Omron CX-Programmer project NewProject (CX-Programmer 9.73)

# PLC NewPLC1: CP1E N60

## Global symbols (name address type ; comment)
0 CHANNEL  ; Timer_2
0.00 BOOL  ; Gripper 1 Unclamp
0.01 BOOL  ; Gripper 1 Clamp
0.02 BOOL  ; Gripper 2 Unclamp
0.03 BOOL  ; Gripper 2 Clamp
0.04 BOOL  ; Rotate CCW
0.05 BOOL  ; Rotate CW
0.06 BOOL  ; Cutting  BWD
0.07 BOOL  ; Cutting FWD
0.08 BOOL  ; Detect component
0.09 BOOL  ; Emergency button
0.10 BOOL  ; Reset button
0.11 BOOL  ; Start Button
100.00 BOOL  ; Grip 1 Clamp/Unclamp
100.01 BOOL  ; Grip 2 Clamp/Unclamp
100.02 BOOL  ; Rotate CW/CCW
100.04 BOOL  ; Blow ON
100.05 BOOL  ; Cutting FWD/BWD
101.00 BOOL  ; Relay Wave Bowl
101.01 BOOL  ; TL GREEN
101.02 BOOL  ; TL RED
101.03 BOOL  ; TL YELLOW
1.00 BOOL  ; Pick Finish
1.01 BOOL  ; rotate finish
1.02 BOOL  ; cut finish
1.11 BOOL  ; Auto mode
20 CHANNEL  ; TIMER_02
200.00 BOOL  ; Gripper 1 Unclamp
200.01 BOOL  ; Gripper 1 Clamp
200.02 BOOL  ; Gripper 2 Unclamp
200.03 BOOL  ; Gripper 2 Clamp
200.04 BOOL  ; Rotate CCW
200.05 BOOL  ; Rotate CW
200.06 BOOL  ; Cutting BWD
200.07 BOOL  ; Cutting FWD
200.08 BOOL  ; Detect Comp
201.00 BOOL  ; Gripper 1
201.01 BOOL  ; Gripper 2
201.02 BOOL  ; Rotate
201.03 BOOL  ; Cutting
201.04 BOOL  ; Manual
201.05 BOOL  ; Auto
201.06 BOOL  ; Emg
201.07 BOOL  ; Start Button
201.08 BOOL  ; Reset Button
201.09 BOOL  ; camera capture
202.00 BOOL  ; Cyl Gripper 1 Clamp/Unclamp
202.01 BOOL  ; Cyl Gripper 2 Clamp/Unclamp
202.02 BOOL  ; Cyl Rotate CW/CCW
202.03 BOOL  ; Blow Bowl ON
202.04 BOOL  ; Cyl Cutting FWD/BWD
202.05 BOOL  ; Process ON
202.06 BOOL  ; Relay Wave ON
203.01 BOOL  ; Camera Capture
203.02 BOOL  ; Move Pick
203.03 BOOL  ; Move Pick Finish
203.04 BOOL  ; move pick finish AR
203.05 BOOL  ; Polarity Result
203.06 BOOL  ; Polarity OK
203.07 BOOL  ; Polarity NG
203.08 BOOL  ; Move to cut
203.09 BOOL  ; Move Cut Finish
203.10 BOOL  ; Move to Pick Finish
203.11 BOOL  ; release cutter
203.12 BOOL  ; capture result
203.13 BOOL  ; Move to Rotate
203.14 BOOL  ; Move to rotate finish
203.15 BOOL  ; Move to Cut after rotate
204.00 BOOL  ; Move to cut after rotate finish
204.01 BOOL  ; Rotate release
205.00 BOOL  ; test
206.00 BOOL  ; Gripper 1 Unclamp
206.01 BOOL  ; Gripper 1 Clamp
206.02 BOOL  ; Gripper 2 Unclamp
206.03 BOOL  ; Gripper 2 Clamp
206.04 BOOL  ; Rotate CCW
206.05 BOOL  ; Rotate CW
206.06 BOOL  ; Cutting BWD
206.07 BOOL  ; Cutting FWD
206.08 BOOL  ; M_Out_Blow
206.09 BOOL  ; m_Detect Comp
206.10 BOOL  ; Bowl Feeder
206.11 BOOL  ; EMG
206.12 BOOL  ; RST
207.00 BOOL  ; Grip 1 Clamp
207.01 BOOL  ; Grip 2 clamp
207.02 BOOL  ; Rotate CW CCW
207.03 BOOL  ; Cutting On
207.04 BOOL  ; Blow On
207.05 BOOL  ; Bowl Feeder
209.01 BOOL  ; TRY LAH
210.00 BOOL  ; pick finish
210.01 BOOL  ; rotate finish
210.02 BOOL  ; cut finish
210.03 BOOL  ; pick move
210.04 BOOL  ; stts pick
210.05 BOOL  ; apalah
210.06 BOOL  ; 1
210.07 BOOL  ; 2
210.08 BOOL  ; stts
210.09 BOOL  ; ok
2.00 BOOL  ; Manual mode
4.00 BOOL  ; Gripper 1 Unclamp
T000 BOOL  ; TIMER_01
T002 BOOL  ; TIMER_02
T003 BOOL  ; Release timer

## Program Auto (cyclic task 0)

### Section PC_INTERFACE

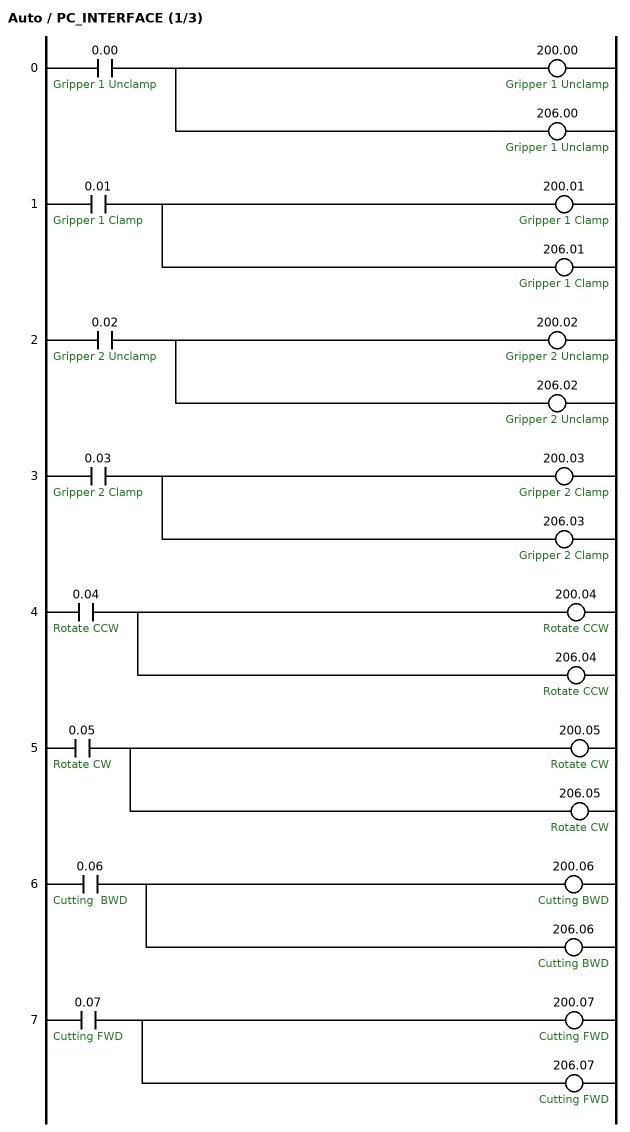
; rung 0
LD 0.00  ; Gripper 1 Unclamp
OUT 200.00  ; Gripper 1 Unclamp
OUT 206.00  ; Gripper 1 Unclamp
; rung 1
LD 0.01  ; Gripper 1 Clamp
OUT 200.01  ; Gripper 1 Clamp
OUT 206.01  ; Gripper 1 Clamp
; rung 2
LD 0.02  ; Gripper 2 Unclamp
OUT 200.02  ; Gripper 2 Unclamp
OUT 206.02  ; Gripper 2 Unclamp
; rung 3
LD 0.03  ; Gripper 2 Clamp
OUT 200.03  ; Gripper 2 Clamp
OUT 206.03  ; Gripper 2 Clamp
; rung 4
LD 0.04  ; Rotate CCW
OUT 200.04  ; Rotate CCW
OUT 206.04  ; Rotate CCW
; rung 5
LD 0.05  ; Rotate CW
OUT 200.05  ; Rotate CW
OUT 206.05  ; Rotate CW
; rung 6
LD 0.06  ; Cutting  BWD
OUT 200.06  ; Cutting BWD
OUT 206.06  ; Cutting BWD
; rung 7
LD 0.07  ; Cutting FWD
OUT 200.07  ; Cutting FWD
OUT 206.07  ; Cutting FWD

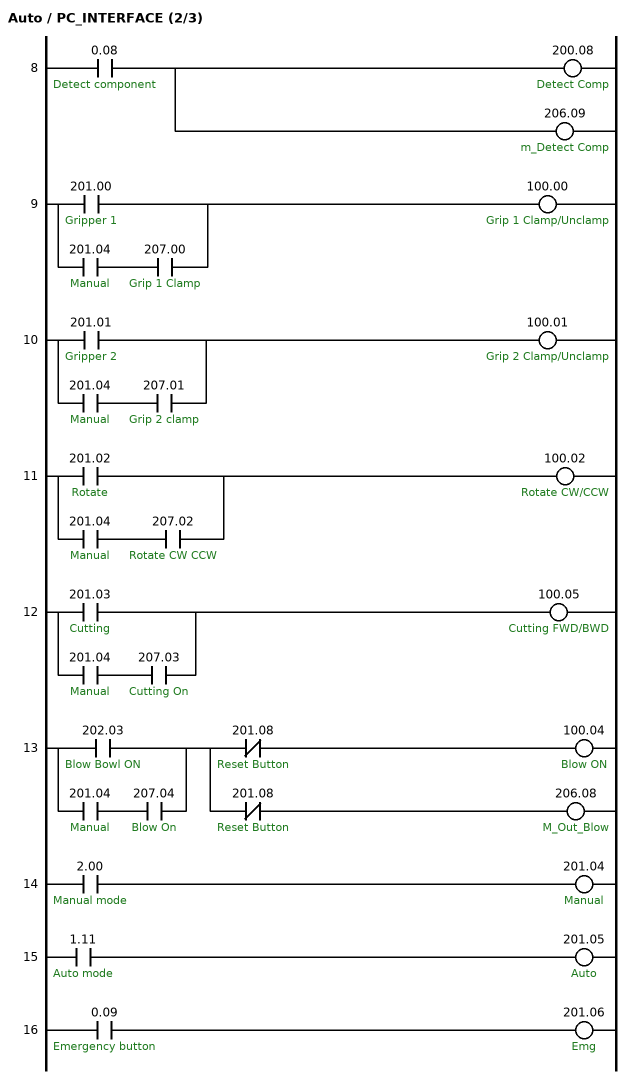
; rung 8
LD 0.08  ; Detect component
OUT 200.08  ; Detect Comp
OUT 206.09  ; m_Detect Comp
; rung 9
LD 201.00  ; Gripper 1
LD 201.04  ; Manual
AND 207.00  ; Grip 1 Clamp
ORLD
OUT 100.00  ; Grip 1 Clamp/Unclamp
; rung 10
LD 201.01  ; Gripper 2
LD 201.04  ; Manual
AND 207.01  ; Grip 2 clamp
ORLD
OUT 100.01  ; Grip 2 Clamp/Unclamp
; rung 11
LD 201.02  ; Rotate
LD 201.04  ; Manual
AND 207.02  ; Rotate CW CCW
ORLD
OUT 100.02  ; Rotate CW/CCW
; rung 12
LD 201.03  ; Cutting
LD 201.04  ; Manual
AND 207.03  ; Cutting On
ORLD
OUT 100.05  ; Cutting FWD/BWD
; rung 13
LD 202.03  ; Blow Bowl ON
LD 201.04  ; Manual
AND 207.04  ; Blow On
ORLD
OUT TR0
ANDNOT 201.08  ; Reset Button
OUT 100.04  ; Blow ON
LD TR0
ANDNOT 201.08  ; Reset Button
OUT 206.08  ; M_Out_Blow
; rung 14
LD 2.00  ; Manual mode
OUT 201.04  ; Manual
; rung 15
LD 1.11  ; Auto mode
OUT 201.05  ; Auto
; rung 16
LD 0.09  ; Emergency button
OUT 201.06  ; Emg

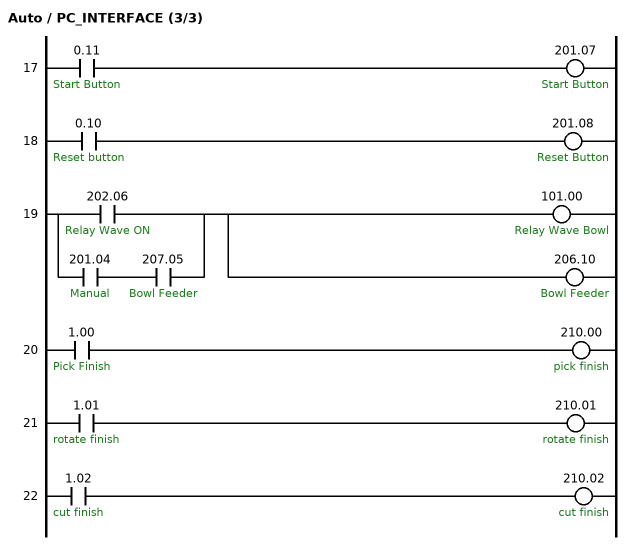
; rung 17
LD 0.11  ; Start Button
OUT 201.07  ; Start Button
; rung 18
LD 0.10  ; Reset button
OUT 201.08  ; Reset Button
; rung 19
LD 202.06  ; Relay Wave ON
LD 201.04  ; Manual
AND 207.05  ; Bowl Feeder
ORLD
OUT 101.00  ; Relay Wave Bowl
OUT 206.10  ; Bowl Feeder
; rung 20
LD 1.00  ; Pick Finish
OUT 210.00  ; pick finish
; rung 21
LD 1.01  ; rotate finish
OUT 210.01  ; rotate finish
; rung 22
LD 1.02  ; cut finish
OUT 210.02  ; cut finish

### Section PROGRAM

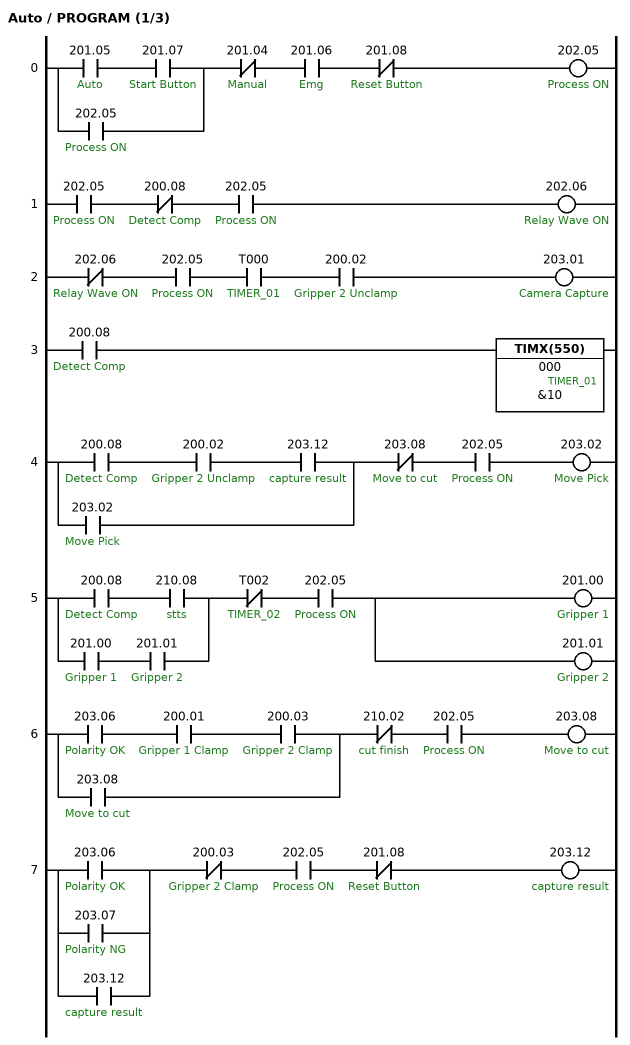
; rung 0
LD 201.05  ; Auto
AND 201.07  ; Start Button
OR 202.05  ; Process ON
ANDNOT 201.04  ; Manual
AND 201.06  ; Emg
ANDNOT 201.08  ; Reset Button
OUT 202.05  ; Process ON
; rung 1
LD 202.05  ; Process ON
ANDNOT 200.08  ; Detect Comp
AND 202.05  ; Process ON
OUT 202.06  ; Relay Wave ON
; rung 2
LDNOT 202.06  ; Relay Wave ON
AND 202.05  ; Process ON
AND T000  ; TIMER_01
AND 200.02  ; Gripper 2 Unclamp
OUT 203.01  ; Camera Capture
; rung 3
LD 200.08  ; Detect Comp
TIMX(550) 000 &10  ; TIMER_01
; rung 4
LD 200.08  ; Detect Comp
AND 200.02  ; Gripper 2 Unclamp
AND 203.12  ; capture result
OR 203.02  ; Move Pick
ANDNOT 203.08  ; Move to cut
AND 202.05  ; Process ON
OUT 203.02  ; Move Pick
; rung 5
LD 200.08  ; Detect Comp
AND 210.08  ; stts
LD 201.00  ; Gripper 1
AND 201.01  ; Gripper 2
ORLD
ANDNOT T002  ; TIMER_02
AND 202.05  ; Process ON
OUT 201.00  ; Gripper 1
OUT 201.01  ; Gripper 2
; rung 6
LD 203.06  ; Polarity OK
AND 200.01  ; Gripper 1 Clamp
AND 200.03  ; Gripper 2 Clamp
OR 203.08  ; Move to cut
ANDNOT 210.02  ; cut finish
AND 202.05  ; Process ON
OUT 203.08  ; Move to cut
; rung 7
LD 203.06  ; Polarity OK
OR 203.07  ; Polarity NG
OR 203.12  ; capture result
ANDNOT 200.03  ; Gripper 2 Clamp
AND 202.05  ; Process ON
ANDNOT 201.08  ; Reset Button
OUT 203.12  ; capture result

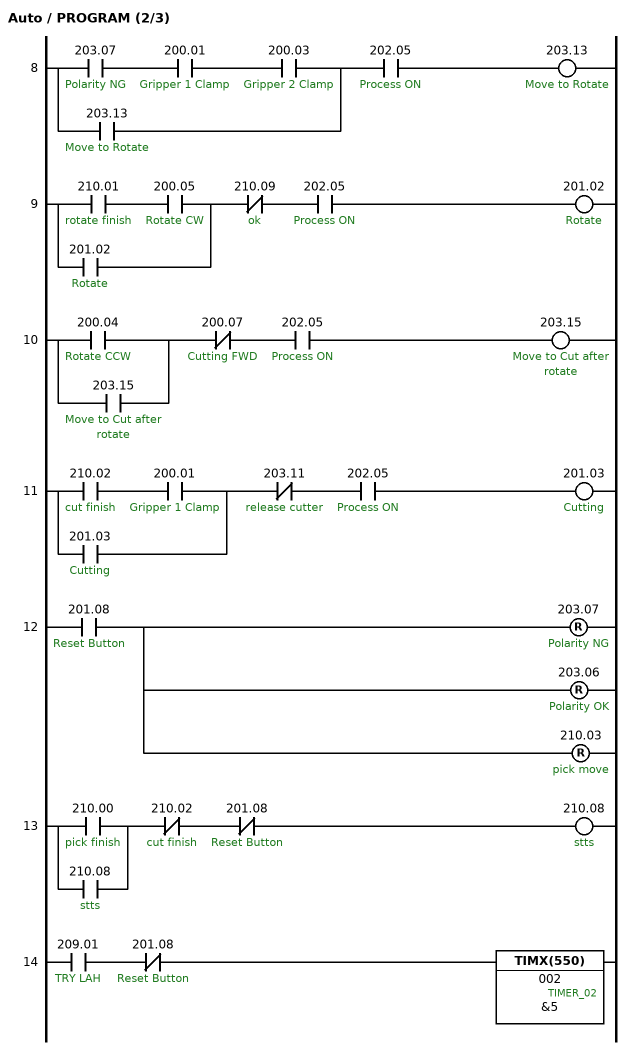
; rung 8
LD 203.07  ; Polarity NG
AND 200.01  ; Gripper 1 Clamp
AND 200.03  ; Gripper 2 Clamp
OR 203.13  ; Move to Rotate
AND 202.05  ; Process ON
OUT 203.13  ; Move to Rotate
; rung 9
LD 210.01  ; rotate finish
AND 200.05  ; Rotate CW
OR 201.02  ; Rotate
ANDNOT 210.09  ; ok
AND 202.05  ; Process ON
OUT 201.02  ; Rotate
; rung 10
LD 200.04  ; Rotate CCW
OR 203.15  ; Move to Cut after rotate
ANDNOT 200.07  ; Cutting FWD
AND 202.05  ; Process ON
OUT 203.15  ; Move to Cut after rotate
; rung 11
LD 210.02  ; cut finish
AND 200.01  ; Gripper 1 Clamp
OR 201.03  ; Cutting
ANDNOT 203.11  ; release cutter
AND 202.05  ; Process ON
OUT 201.03  ; Cutting
; rung 12
LD 201.08  ; Reset Button
RSET 203.07  ; Polarity NG
RSET 203.06  ; Polarity OK
RSET 210.03  ; pick move
; rung 13
LD 210.00  ; pick finish
OR 210.08  ; stts
ANDNOT 210.02  ; cut finish
ANDNOT 201.08  ; Reset Button
OUT 210.08  ; stts
; rung 14
LD 209.01  ; TRY LAH
ANDNOT 201.08  ; Reset Button
TIMX(550) 002 &5  ; TIMER_02

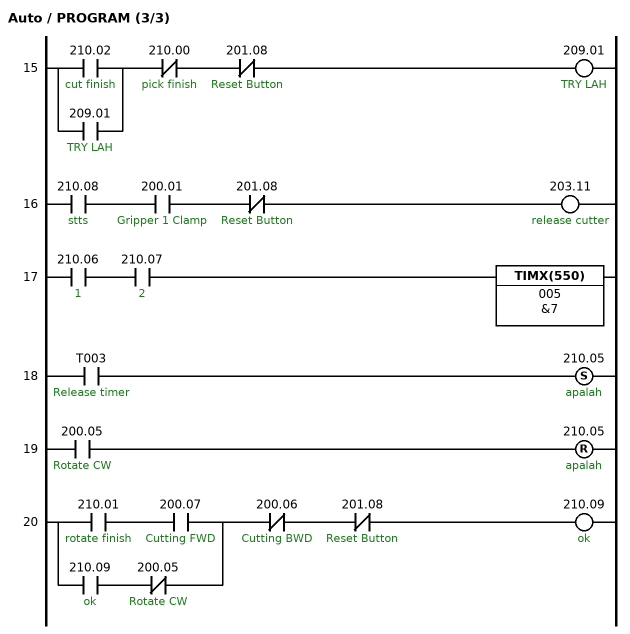
; rung 15
LD 210.02  ; cut finish
OR 209.01  ; TRY LAH
ANDNOT 210.00  ; pick finish
ANDNOT 201.08  ; Reset Button
OUT 209.01  ; TRY LAH
; rung 16
LD 210.08  ; stts
AND 200.01  ; Gripper 1 Clamp
ANDNOT 201.08  ; Reset Button
OUT 203.11  ; release cutter
; rung 17
LD 210.06  ; 1
AND 210.07  ; 2
TIMX(550) 005 &7
; rung 18
LD T003  ; Release timer
SET 210.05  ; apalah
; rung 19
LD 200.05  ; Rotate CW
RSET 210.05  ; apalah
; rung 20
LD 210.01  ; rotate finish
AND 200.07  ; Cutting FWD
LD 210.09  ; ok
ANDNOT 200.05  ; Rotate CW
ORLD
ANDNOT 200.06  ; Cutting BWD
ANDNOT 201.08  ; Reset Button
OUT 210.09  ; ok

### Section Status

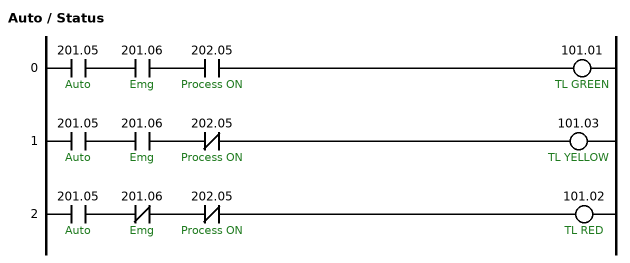
; rung 0
LD 201.05  ; Auto
AND 201.06  ; Emg
AND 202.05  ; Process ON
OUT 101.01  ; TL GREEN
; rung 1
LD 201.05  ; Auto
AND 201.06  ; Emg
ANDNOT 202.05  ; Process ON
OUT 101.03  ; TL YELLOW
; rung 2
LD 201.05  ; Auto
ANDNOT 201.06  ; Emg
ANDNOT 202.05  ; Process ON
OUT 101.02  ; TL RED

### Section END
; rung 0
END(001)